(* Logix 5000 project; controller UniStream_COMM vendor 1 type 14 code 96 rev 32.11; software revision 32.00 *)

TASK MainTask (continuous, watchdog 500 ms) : MainProgram

MODULES
   Local : vendor 1 type 14 code 96 (ICP 0, rev 32.11)
      ENBT : 1756-ENBT (ICP 2, Ethernet 192.168.1.249, rev 4.3)
         UniStream : ETHERNET-MODULE (Ethernet 192.168.1.251, rev 1.1, Output RPI 1500 ms)
END_MODULES

TYPE EIP_Data :
STRUCT
   Reales : REAL[4];
   Bits : BOOL[32];
   Int16 : INT[4];
   Int32 : DINT[4];
END_STRUCT
END_TYPE

VAR_GLOBAL   (* controller tags *)
   EIP_Read : EIP_Data := (Reales[0] := 12.2, Reales[3] := 15.5, Bits[0] := 1, Bits[8] := 1, Bits[30] := 1, Int16[0] := 40, Int16[3] := 43, Int32[0] := 4321, Int32[3] := 1234);
   EIP_Write : EIP_Data := (Reales[0] := 11.22, Reales[1] := 22.33, Reales[2] := 33.44, Reales[3] := 44.55, Bits[0] := 1, Bits[1] := 1, Bits[29] := 1, Bits[30] := 1, Int16[0] := 1601, Int16[1] := 1602, Int16[2] := 1603, Int16[3] := 1604, Int32[0] := 3201, Int32[1] := 3202, Int32[2] := 3203, Int32[3] := 3204);
END_VAR

PROGRAM MainProgram   (* main routine MainRoutine *)

ROUTINE MainRoutine   (* ladder *)
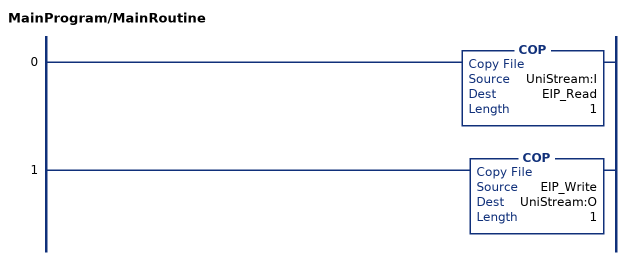
   0: COP(UniStream:I,EIP_Read,1);
   1: COP(EIP_Write,UniStream:O,1);
END_ROUTINE
END_PROGRAM
